(* Logix 5000 project; controller ChemicalProcess Emulate 5570 rev 30.12; software revision 30.02 *)

TASK MainTask (continuous, watchdog 500 ms) : MainProgram

MODULES
   Local : Emulate 5570 (ICP 3, rev 30.12)
      IO4 : vendor 1 type 0 code 15 (ICP 4, rev 1.1, Output RPI 15 ms)
      IO8 : vendor 1 type 0 code 15 (ICP 8, rev 1.1, Output RPI 15 ms)
END_MODULES

VAR_GLOBAL   (* controller tags *)
   auxillaryContact : BOOL;
   DrainState : BOOL;
   MixerState : BOOL;
   motorTimer : TIMER := (PRE := 30);
   StartONS : BOOL;
   step : DINT;
   Valve1LimitSwitch : BOOL;   // Limit switch that turns on if the valve is fully open.
   Valve2LimitSwitch : BOOL;   // Limit switch that turns on if the valve is fully open.
   Valve3LimitSwitch : BOOL;   // Limit switch that turns on if the valve is fully open.
END_VAR

PROGRAM MainProgram   (* main routine MainRoutine *)
VAR
   DrainStart : BOOL;
   DrainStop : BOOL;
   Feed1Start : BOOL;
   Feed1State : BOOL;
   Feed1Stop : BOOL;
   Feed2Start : BOOL;
   Feed2State : BOOL;
   Feed2Stop : BOOL;
   MixerStart : BOOL;
   MixerStop : BOOL;
   Motor1Out : ALIAS FOR Local:8:O.Data[0].3;   // Output bit that controls the motor. On = motor commanded on.
   SensorLevel1 : ALIAS FOR Local:4:I.Data[0].12;   // On = at or above level 1. Off = at or below level 1.
   SensorLevel2 : ALIAS FOR Local:4:I.Data[0].13;   // On = at or above level 2. Off = at or below level 2.
   SensorTankEmpty : ALIAS FOR Local:4:I.Data[0].14;   // On = tank empty. Off = tank not empty.
   Start : ALIAS FOR Local:4:I.Data[0].0;   // Starts the chemical process.
   Valve1Out : ALIAS FOR Local:8:O.Data[0].1;   // Output bit that controls the valve. On = valve commanded open.
   Valve2Out : ALIAS FOR Local:8:O.Data[0].2;   // Output bit that controls the valve. On = valce commanded open.
   Valve3Out : ALIAS FOR Local:8:O.Data[0].1;   // Output bit that controls the valve. On = valve commanded open.
END_VAR

ROUTINE Drain   (* ladder *)
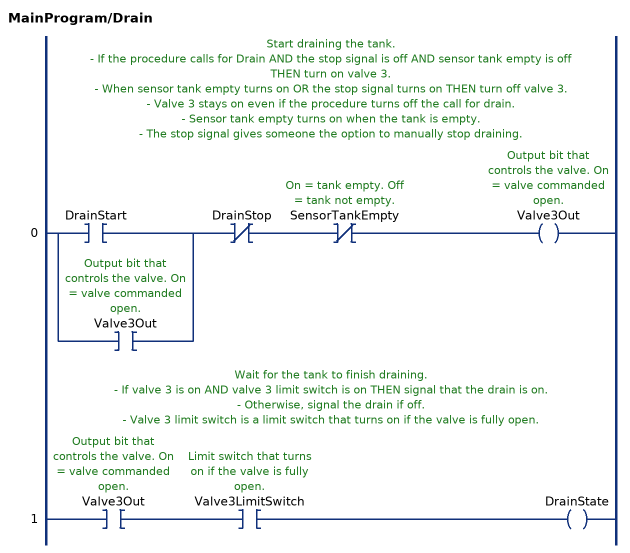
   // Start draining the tank.
   // - If the procedure calls for Drain AND the stop signal is off AND sensor tank empty is off THEN turn on valve 3.
   // - When sensor tank empty turns on OR the stop signal turns on THEN turn off valve 3.
   // - Valve 3 stays on even if the procedure turns off the call for drain.
   // - Sensor tank empty turns on when the tank is empty.
   // - The stop signal gives someone the option to manually stop draining.
   0: [XIC(DrainStart) ,XIC(Valve3Out) ]XIO(DrainStop)XIO(SensorTankEmpty)OTE(Valve3Out);
   // Wait for the tank to finish draining.
   // - If valve 3 is on AND valve 3 limit switch is on THEN signal that the drain is on.
   // - Otherwise, signal the drain if off.
   // - Valve 3 limit switch is a limit switch that turns on if the valve is fully open.
   1: XIC(Valve3Out)XIC(Valve3LimitSwitch)OTE(DrainState);
END_ROUTINE

ROUTINE Fill_Chemical_1   (* ladder *)
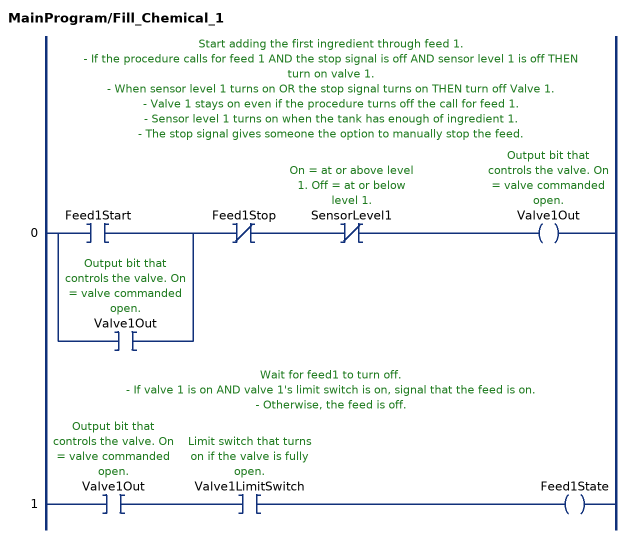
   // Start adding the first ingredient through feed 1.
   // - If the procedure calls for feed 1 AND the stop signal is off AND sensor level 1 is off THEN turn on valve 1.
   // - When sensor level 1 turns on OR the stop signal turns on THEN turn off Valve 1.
   // - Valve 1 stays on even if the procedure turns off the call for feed 1.
   // - Sensor level 1 turns on when the tank has enough of ingredient 1.
   // - The stop signal gives someone the option to manually stop the feed.
   0: [XIC(Feed1Start) ,XIC(Valve1Out) ]XIO(Feed1Stop)XIO(SensorLevel1)OTE(Valve1Out);
   // Wait for feed1 to turn off.
   // - If valve 1 is on AND valve 1's limit switch is on, signal that the feed is on.
   // - Otherwise, the feed is off.
   1: XIC(Valve1Out)XIC(Valve1LimitSwitch)OTE(Feed1State);
END_ROUTINE

ROUTINE Fill_Chemical_2   (* ladder *)
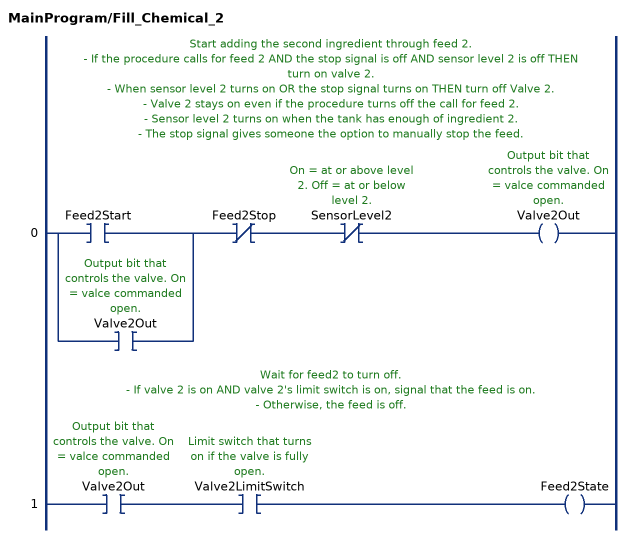
   // Start adding the second ingredient through feed 2.
   // - If the procedure calls for feed 2 AND the stop signal is off AND sensor level 2 is off THEN turn on valve 2.
   // - When sensor level 2 turns on OR the stop signal turns on THEN turn off Valve 2.
   // - Valve 2 stays on even if the procedure turns off the call for feed 2.
   // - Sensor level 2 turns on when the tank has enough of ingredient 2.
   // - The stop signal gives someone the option to manually stop the feed.
   0: [XIC(Feed2Start) ,XIC(Valve2Out) ]XIO(Feed2Stop)XIO(SensorLevel2)OTE(Valve2Out);
   // Wait for feed2 to turn off.
   // - If valve 2 is on AND valve 2's limit switch is on, signal that the feed is on.
   // - Otherwise, the feed is off.
   1: XIC(Valve2Out)XIC(Valve2LimitSwitch)OTE(Feed2State);
END_ROUTINE

ROUTINE MainRoutine   (* ladder *)
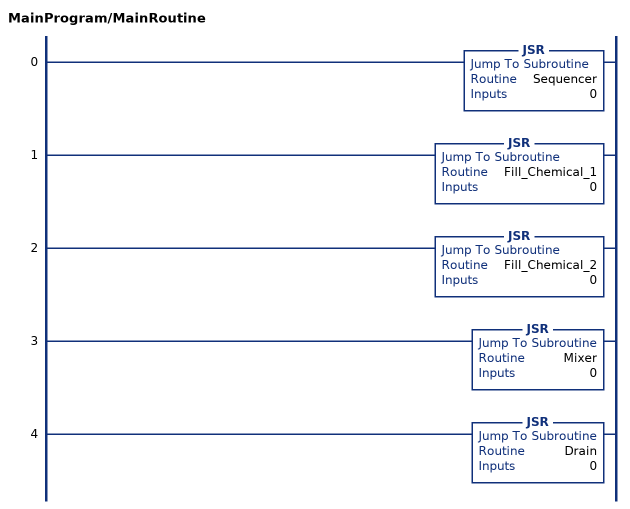
   0: JSR(Sequencer,0);
   1: JSR(Fill_Chemical_1,0);
   2: JSR(Fill_Chemical_2,0);
   3: JSR(Mixer,0);
   4: JSR(Drain,0);
END_ROUTINE

ROUTINE Mixer   (* ladder *)
// Mix ingredients
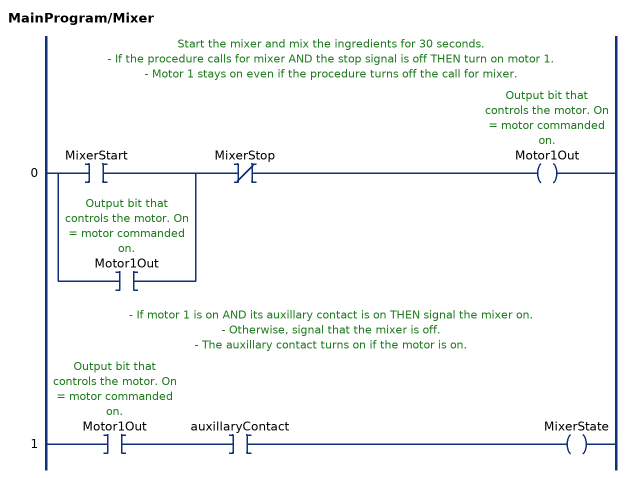
   // Start the mixer and mix the ingredients for 30 seconds.
   // - If the procedure calls for mixer AND the stop signal is off THEN turn on motor 1.
   // - Motor 1 stays on even if the procedure turns off the call for mixer.
   0: [XIC(MixerStart) ,XIC(Motor1Out) ]XIO(MixerStop)OTE(Motor1Out);
   // - If motor 1 is on AND its auxillary contact is on THEN signal the mixer on.
   // - Otherwise, signal that the mixer is off.
   // - The auxillary contact turns on if the motor is on.
   1: XIC(Motor1Out)XIC(auxillaryContact)OTE(MixerState);
END_ROUTINE

ROUTINE Sequencer   (* ladder *)
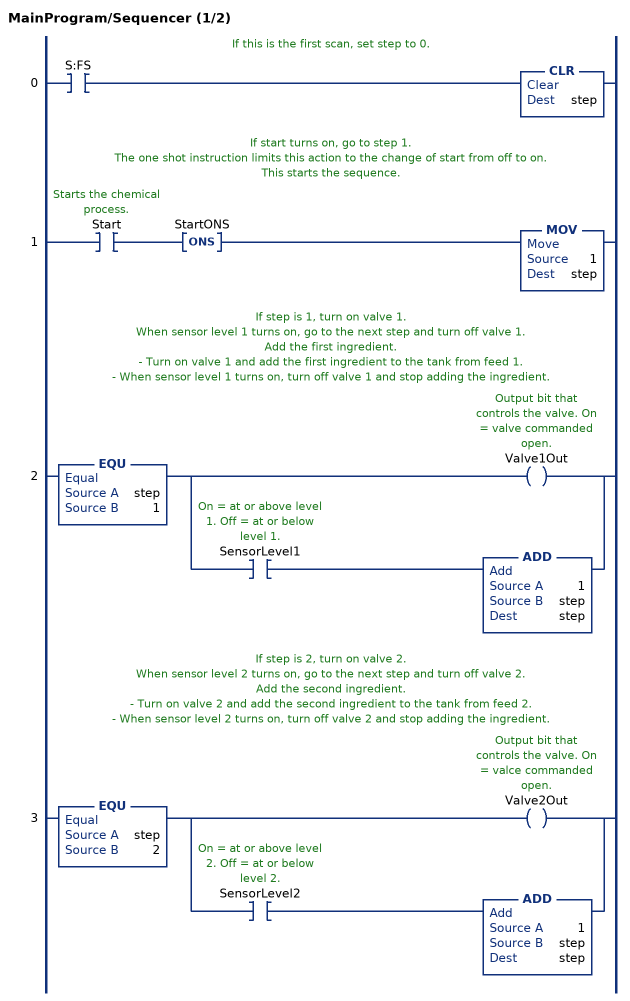
   // If this is the first scan, set step to 0.
   0: XIC(S:FS)CLR(step);
   // If start turns on, go to step 1.
   // The one shot instruction limits this action to the change of start from off to on.
   // This starts the sequence.
   1: XIC(Start)ONS(StartONS)MOV(1,step);
   // If step is 1, turn on valve 1.
   // When sensor level 1 turns on, go to the next step and turn off valve 1.
   // Add the first ingredient.
   // - Turn on valve 1 and add the first ingredient to the tank from feed 1.
   // - When sensor level 1 turns on, turn off valve 1 and stop adding the ingredient.
   2: EQU(step,1)[OTE(Valve1Out) ,XIC(SensorLevel1) ADD(1,step,step) ];
   // If step is 2, turn on valve 2.
   // When sensor level 2 turns on, go to the next step and turn off valve 2.
   // Add the second ingredient.
   // - Turn on valve 2 and add the second ingredient to the tank from feed 2.
   // - When sensor level 2 turns on, turn off valve 2 and stop adding the ingredient.
   3: EQU(step,2)[OTE(Valve2Out) ,XIC(SensorLevel2) ADD(1,step,step) ];
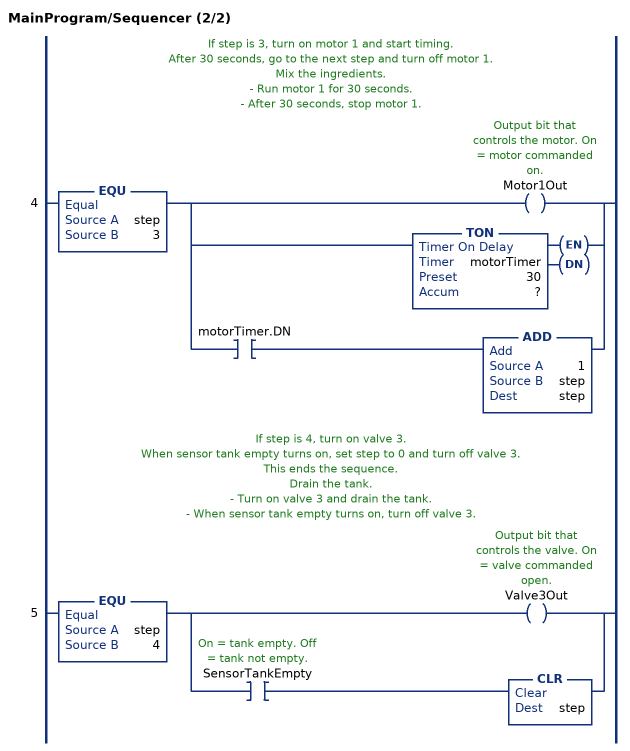
   // If step is 3, turn on motor 1 and start timing.
   // After 30 seconds, go to the next step and turn off motor 1.
   // Mix the ingredients.
   // - Run motor 1 for 30 seconds.
   // - After 30 seconds, stop motor 1.
   4: EQU(step,3)[OTE(Motor1Out) ,[TON(motorTimer,?,?) ,XIC(motorTimer.DN) ADD(1,step,step) ] ];
   // If step is 4, turn on valve 3.
   // When sensor tank empty turns on, set step to 0 and turn off valve 3.
   // This ends the sequence.
   // Drain the tank.
   // - Turn on valve 3 and drain the tank.
   // - When sensor tank empty turns on, turn off valve 3.
   5: EQU(step,4)[OTE(Valve3Out) ,XIC(SensorTankEmpty) CLR(step) ];
END_ROUTINE
END_PROGRAM
